FUNCTION_BLOCK FB_Ctrl_Cam IMPLEMENTS I_Cam_Ctrl
VAR_INPUT
END_VAR
VAR_OUTPUT
END_VAR
VAR
  _bInSync,
  _bBusy,
  _bError         : BOOL;

  _udiError       : UDINT;

  _pAxisSlave,
  _pAxisMaster    : POINTER TO Tc2_MC2.AXIS_REF;  

  _fbCamIn        : Tc2_MC2_Camming.MC_CamIn_V2;
  _fbCamOut       : Tc2_MC2_Camming.MC_CamOut;

END_VAR

METHOD CamIn : BOOL
VAR_INPUT
  bExecute      : BOOL;
  stCamIn       : ST_CamIn;
END_VAR
VAR_INST
  _nState       : UINT;

END_VAR
IF NOT (_pAxisMaster <> 0) OR
   NOT (_pAxisSlave <> 0)
THEN
  RETURN;
END_IF

IF NOT bExecute
THEN
  _nState         := 0;
END_IF

CASE _nState 
OF
  0:
    _fbCamIn(
          Master              := _pAxisMaster^, 
          Slave               := _pAxisSlave^, 
          Execute             := FALSE, 
          ActivationMode      := stCamIn.StartMode, 
          ActivationPosition:= , 
          CamTableID:= , 
          Scaling:= , 
          Options:= , 
          InSync=> , 
          Busy=> , 
          Active=> , 
          CommandAborted=> , 
          Error=> , 
          ErrorID=> );


END_CASE
END_METHOD

PROPERTY MasterAxis : POINTER TO Tc2_MC2.AXIS_REF
SET
_pAxisMaster := MasterAxis;
END_SET
END_PROPERTY

PROPERTY SlaveAxis : POINTER TO Tc2_MC2.AXIS_REF
SET
	_pAxisSlave := SlaveAxis;
END_SET
END_PROPERTY

END_FUNCTION_BLOCK

(* stored: Version 1.1.0.1, ProductVersion 3.1.4024.12
   POU FB_Ctrl_Cam: Id {ec589a30-c0cb-07ed-066e-6383c15441f2}, SpecialFunc None
   Method CamIn: Id {3f9750f1-fba9-0a95-0065-08ee42705959}
   Property MasterAxis: Id {e9ea0207-855a-0548-0716-961e2367e1ea}
   Set Set: Id {0a9470a5-2a30-0d8f-36f1-350a54b8ca71}
   Property SlaveAxis: Id {2852ae05-60dc-06b3-3437-9244c97fcebd}
   Set Set: Id {f7a3f116-7de2-069b-015b-1b5ea80624b7} *)
